FUNCTION_BLOCK PUBLIC FB_StepWorker IMPLEMENTS I_StepWorker
VAR_INPUT
	bResetTimeout : BOOL;
END_VAR
VAR_OUTPUT
	uiStep : UINT;
	bTimeout : BOOL;
END_VAR
VAR
	uiConditionCounter : UINT := 1;
	aConditions	: ARRAY[1..cMaxConditions] OF I_StepCondition;

	bTimeoutFlag : BOOL;	
	fbTimeout : TON;
	fbTimer : TON;
	tTimeIntern : TIME;
END_VAR
VAR CONSTANT
	cMaxConditions : UINT := 25;
	
END_VAR

IF bResetTimeout
THEN
	bResetTimeout := FALSE;
	bTimeout := FALSE;
	bTimeoutFlag := FALSE;
END_IF

fbTimeout(IN:=bTimeoutFlag, PT:=tTimeIntern , Q=>bTimeout);
fbTimer();

METHOD AndNegCondition : I_StepWorker
VAR_INPUT
	itfStepCondition : I_StepCondition;
END_VAR
VAR
	i : UINT;
END_VAR
andNegCondition := THIS^;
IF itfStepCondition = 0 //Avoid null pointer exception.
	OR uiConditionCounter = cMaxConditions + 1
THEN
	
	RETURN;
END_IF

FOR i := 1 TO uiConditionCounter DO
	IF aConditions[i] = itfStepCondition 
	THEN
		//Condition already added.
		RETURN;
	END_IF
END_FOR
 
//Add new condition.
itfStepCondition.NegCondition();
aConditions[uiConditionCounter] := itfStepCondition;
uiConditionCounter := uiConditionCounter + 1;
END_METHOD

METHOD AndPosCondition : I_StepWorker
VAR_INPUT
	itfStepCondition : I_StepCondition;
END_VAR
VAR
	i : UINT;
END_VAR
andPosCondition := THIS^;
IF itfStepCondition = 0 //Avoid null pointer exception.
	OR uiConditionCounter = cMaxConditions + 1
THEN
	
	RETURN;
END_IF

FOR i := 1 TO uiConditionCounter DO
	IF aConditions[i] = itfStepCondition 
	THEN
		//Condition already added.
		RETURN;
	END_IF
END_FOR
 
//Add new condition.
itfStepCondition.PosCondition();
aConditions[uiConditionCounter] := itfStepCondition;
uiConditionCounter := uiConditionCounter + 1;
END_METHOD

METHOD NextStep : UINT
VAR_INPUT
	uiNextStep : UINT;
END_VAR
VAR
	i : UINT;
END_VAR
IF bTimeout
THEN
	NextStep := uiStep;
	RETURN;
END_IF
	
FOR i := 1 TO (uiConditionCounter-1) DO
	IF aConditions[i].isNegative
	THEN
		IF aConditions[i].getValue = TRUE 
		THEN
			//one Condition is True therefor exit.
			NextStep := uiStep;
			RETURN;
		END_IF
	ELSIF aConditions[i].isPositive
	THEN
		IF aConditions[i].getValue = FALSE 
		THEN
			//one Condition is false therefor exit.
			NextStep := uiStep;
			RETURN;
		END_IF
	END_IF
	
	
END_FOR

//All conditions met
bTimeoutFlag := FALSE;

//Reset the condition counter and conditions
FOR i := 1 TO (uiConditionCounter-1) DO
	aConditions[i] := 0;
END_FOR

uiConditionCounter := 1;

IF fbTimer.IN 
	AND fbTimer.Q
THEN
	fbTimer.IN := FALSE;
	uiStep := uiNextStep;
	NextStep := uiNextStep;
ELSIF fbTimer.IN
	AND NOT fbTImer.Q
THEN
	NextStep := uiStep;
ELSE
	uiStep := uiNextStep;
	NextStep := uiNextStep;	
END_IF
END_METHOD

METHOD SetTimeout : I_StepWorker
VAR_INPUT
	tTime : TIME;
END_VAR
SetTimeout := THIS^;
tTimeIntern := tTime;
bTimeoutFlag := TRUE;
END_METHOD

METHOD SetTimer : I_StepWorker
VAR_INPUT
	tTime : TIME;
END_VAR
SetTimer := THIS^;
fbTimer.PT := tTime;
fbTimer.IN := TRUE;
END_METHOD

END_FUNCTION_BLOCK

(* stored: Version 1.1.0.1, ProductVersion 3.1.4024.2
   POU FB_StepWorker: Id {44f74475-c942-48f3-81b1-525d23658d36}, SpecialFunc None
   Method AndNegCondition: Id {6f316bf1-42e4-4e90-a61a-7baff43334c0}
   Method AndPosCondition: Id {8ec1ae46-390d-491a-806a-a2abcd8e50a5}
   Method NextStep: Id {fbdecb39-2f5a-4df6-a2c8-cb28af62eebe}
   Method SetTimeout: Id {fe6f174f-06ef-4ced-b025-bdae118f56fe}
   Method SetTimer: Id {feb9bbef-be60-4033-bb9b-8d4f4516e849} *)
